(* CoDeSys 2.3 export: WRITEOUTPUTS.EXP *)

(* POU InputsOutputs/WriteOutputs, FBD *)
PROGRAM WriteOutputs
VAR_INPUT
	OUT0: BOOL;
	OUT1: BOOL;
	OUT2: BOOL;
	OUT3: BOOL;
	OUT4: BOOL;
	OUT5: BOOL;
	OUT6: BOOL;
	OUT7: BOOL;
END_VAR
VAR
	_output: ARRAY[0..7] OF OUTPUT;
END_VAR
VAR CONSTANT
	ModeOutput_Off: BYTE := 0;
	ModeOutput_HighSide: BYTE := 2;
	ModeOutput_HighSide_Diag: BYTE := 15;
	ModeOutput_HighSide_Diag_Protection: BYTE := 16;
END_VAR
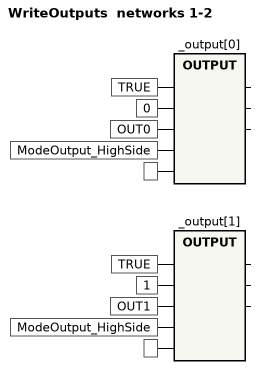
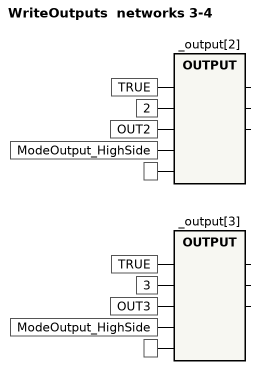
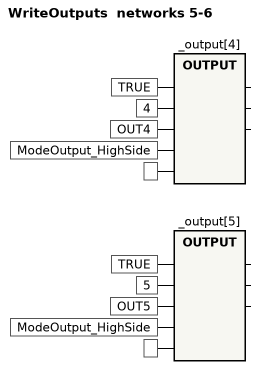
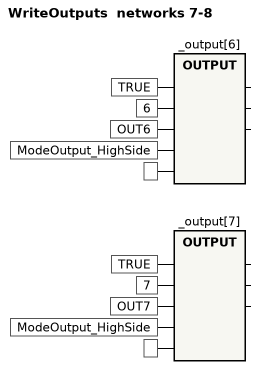
_FBD_ (* Function Block Diagram *)
NETWORK 1
	_output[0]:OUTPUT(TRUE, 0, OUT0, ModeOutput_HighSide, )
NETWORK 2
	_output[1]:OUTPUT(TRUE, 1, OUT1, ModeOutput_HighSide, )
NETWORK 3
	_output[2]:OUTPUT(TRUE, 2, OUT2, ModeOutput_HighSide, )
NETWORK 4
	_output[3]:OUTPUT(TRUE, 3, OUT3, ModeOutput_HighSide, )
NETWORK 5
	_output[4]:OUTPUT(TRUE, 4, OUT4, ModeOutput_HighSide, )
NETWORK 6
	_output[5]:OUTPUT(TRUE, 5, OUT5, ModeOutput_HighSide, )
NETWORK 7
	_output[6]:OUTPUT(TRUE, 6, OUT6, ModeOutput_HighSide, )
NETWORK 8
	_output[7]:OUTPUT(TRUE, 7, OUT7, ModeOutput_HighSide, )
_END_FBD_
END_PROGRAM
